// TwinCAT 3 PLC project motion_abstraction_sample
// ProgramVersion: 3.1.4026.17
// libraries:
//   LCLS General, * (SLAC)
//   LCLS_OOPMotion, * (SLAC)
//   Tc2_MC2, * (Beckhoff Automation GmbH)
//   Tc2_NC, * (Beckhoff Automation GmbH)
//   Tc2_Standard, * (Beckhoff Automation GmbH)
//   Tc2_System, * (Beckhoff Automation GmbH)
// project tree:
//   DUTs/ ENUM_AxisStates.TcDUT (not stored)
//   GVLs/ GVL_Axes.TcGVL
//   / PlcTask.TcTTO
//   POUs/ MAIN.TcPOU
// real-time tasks:
//   TASK PlcTask: cycle T#10ms, priority 20, ADS port 350
// motion (NC):
//   TASK NC-Task 1 SAF: cycle T#2ms, priority 4, ADS port 501
//   TASK NC-Task 1 SVB: cycle T#10ms, priority 8, ADS port 511
//   AXIS Axis 4 (id 4)
//     OtherSettings: AllowMotionCmdToSlave=true
//     encoder EncType=1
//     drive DrvType=5
//       Analog: TorqueSetpointScale=10, ScaleFactorActTorque=0.1
//       TimeComp: TaskDelayCycles=1
//     controller CtrType=1
//       CtrPara: PriorControlFactor=1
//         Observer: BandWidth=20
//   AXIS Axis 3 (id 3)
//     OtherSettings: AllowMotionCmdToSlave=true
//     encoder EncType=1
//     drive DrvType=5
//       Analog: TorqueSetpointScale=10, ScaleFactorActTorque=0.1
//       TimeComp: TaskDelayCycles=1
//     controller CtrType=1
//       CtrPara: PriorControlFactor=1
//         Observer: BandWidth=20
//   AXIS Axis 2 (id 2)
//     OtherSettings: AllowMotionCmdToSlave=true
//     encoder EncType=1
//     drive DrvType=5
//       Analog: TorqueSetpointScale=10, ScaleFactorActTorque=0.1
//       TimeComp: TaskDelayCycles=1
//     controller CtrType=1
//       CtrPara: PriorControlFactor=1
//         Observer: BandWidth=20
//   AXIS Axis 1 (id 1)
//     OtherSettings: AllowMotionCmdToSlave=true
//     encoder EncType=1
//       ActPosCorrection: Enable=true
//     drive DrvType=5
//       Analog: TorqueSetpointScale=10, ScaleFactorActTorque=0.1
//       TimeComp: TaskDelayCycles=1
//     controller CtrType=1
//       CtrPara: PriorControlFactor=1
//         Observer: BandWidth=20
// variable links:
//   motion_abstraction_sample Instance <-> NC-Task 1 SAF/Axes/Axis 1
//     PlcTask Inputs/GVL_Axes.Axes[1].NcToPlc <-> Outputs/ToPlc
//     PlcTask Outputs/GVL_Axes.Axes[1].PlcToNc <-> Inputs/FromPlc
//   motion_abstraction_sample Instance <-> NC-Task 1 SAF/Axes/Axis 2
//     PlcTask Inputs/GVL_Axes.Axes[2].NcToPlc <-> Outputs/ToPlc
//     PlcTask Outputs/GVL_Axes.Axes[2].PlcToNc <-> Inputs/FromPlc
//   motion_abstraction_sample Instance <-> NC-Task 1 SAF/Axes/Axis 3
//     PlcTask Inputs/GVL_Axes.Axes[3].NcToPlc <-> Outputs/ToPlc
//     PlcTask Outputs/GVL_Axes.Axes[3].PlcToNc <-> Inputs/FromPlc
//   motion_abstraction_sample Instance <-> NC-Task 1 SAF/Axes/Axis 4
//     PlcTask Inputs/GVL_Axes.Axes[4].NcToPlc <-> Outputs/ToPlc
//     PlcTask Outputs/GVL_Axes.Axes[4].PlcToNc <-> Inputs/FromPlc

CONFIGURATION motion_abstraction_sample
    RESOURCE PLC ON TwinCAT3
        TASK PlcTask(INTERVAL := T#10ms, PRIORITY := 20);
        PROGRAM MAIN WITH PlcTask : MAIN;
    END_RESOURCE
END_CONFIGURATION

// ---- GVLs/GVL_Axes.TcGVL
{attribute 'qualified_only'}
VAR_GLOBAL
    Axes :  ARRAY[1..4] OF AXIS_REF;
END_VAR

// ---- POUs/MAIN.TcPOU
PROGRAM MAIN
VAR
    fbPersistentDataStorage : FB_PersistentDataStorage;
	{attribute 'pytmc' := '
		axis-link: GVL_Axes.Axes[1]
		pv: TST:MOTION:SLITX
	'}
   	slitX : FB_MotionStageNC(	sName := 'slitX',
                                        AxisRef := GVL_Axes.Axes[1],
                                        iPersistentDataStorage := fbPersistentDataStorage
                                    ) ;
	{attribute 'pytmc' := '
		axis-link: GVL_Axes.Axes[2]
		pv: TST:MOTION:SLITY
	'}
   	slitY : FB_MotionStageNC(	sName := 'slitY',
                                        AxisRef := GVL_Axes.Axes[2],
                                        iPersistentDataStorage := fbPersistentDataStorage
                                    ) := (EnableMode:=E_StageEnableMode.ALWAYS);
	{attribute 'pytmc' := '
		axis-link: GVL_Axes.Axes[3]
		pv: TST:MOTION:SLITZ
	'}
   	slitZ : FB_MotionStageNC(	sName := 'slitZ',
                                        AxisRef := GVL_Axes.Axes[3],
                                        iPersistentDataStorage := fbPersistentDataStorage
                                    ) ;
   	dummy : FB_MotionStageNC(	sName := 'dummy',
                                        AxisRef := GVL_Axes.Axes[4],
                                        iPersistentDataStorage := fbPersistentDataStorage
                                    ) ;
END_VAR

fbPersistentDataStorage();
slitX();
slitY();
slitZ();
dummy();

END_PROGRAM
